{attribute 'qualified_only'}
{attribute 'strict'}
TYPE E_SlitPairStates :
(
    eInit := 0,
    eEnableRealGenerators,
    eDisableRealGenerators,
    eEnableVirtualGenerators,
    eDisableVirtualGenerators,
    eWaitForVirtualMoveDone,
    eWaitForRealMoveDone,
    eError,
    eOperational,
    eWaitForVirtualHomed,
    eWaitForRealHomed,
    eCheckRealAxisGeneratorsEnabled,
    eCheckVirtualAxisGeneratorsEnabled,
    eDisableGenerators
);
END_TYPE

(* stored: Version 1.1.0.1, ProductVersion 3.1.4024.11
   DUT E_SlitPairStates: Id {6665fbaf-b520-47d5-8ce7-9872d8af20f7} *)
